Universal Robots PolyScope program: 1tra2.urp

Program 1tra2 (installation=default directory=/home/ur/ursim-current/programs createdIn=5.12.6.1102099 lastSavedIn=5.12.6.1102099 robotSerialNumber=20195599999)
Calibrated DH parameters: a=[0, -0.425, -0.3922, 0, 0, 0]; d=[0.1625, 0, 0, 0.1333, 0.0997, 0.0996]; alpha=[1.570796, 0, 0, 1.570796, -1.570796, 0]; deltaTheta=[0, 0, 0, 0, 0, 0]
Robot Program (runOnlyOnce=false)
  Set DigitalOutput pin=digital_out[0]; digitalValue=1
  Popup Message (haltProgram=false message=and inputType=Text)
  Wait Sleep waitTime=5
  URCap External Control (External Control, FZI Research Center for Information Technology)
